// TIA Portal V16 export
// export: Created 2023-03-29T11:03:25.0566469Z, ExportSetting WithDefaults, DisplayName Totally Integrated Automation Portal, DisplayVersion V16 Update 6, DisplayName TIA Portal Version Control Interface, DisplayVersion V16 Update 2, DisplayName TIA Portal Openness, DisplayVersion V16 Update 6, DisplayName STEP 7 Professional, DisplayVersion V16 Update 6, DisplayName STEP 7 Safety, DisplayVersion V16, DisplayName WinCC Advanced, DisplayVersion V16 Update 6
FUNCTION_BLOCK "Client_ModbusTCP_read_control"   // FB1, LAD
TITLE = Pobieranie parametrów sterowania
{ S7_Optimized_Access := 'TRUE' }
AUTHOR : rtecmer
VERSION : 0.1
// funkcja pobiera z servera dane przekazywanie z PLC 1 do kontroli systemu
// stored: AutoNumber true, IsIECCheckEnabled false, IsRetainMemResEnabled false, MemoryReserve 250, SetENOAutomatically false, UDAEnableTagReadback false
   VAR_IN_OUT
      modbustcp_przetwarzanie_In : Bool;
      modbustcp_przetwarzanie_out : Bool;
   END_VAR
   VAR_TEMP   // added for the SCL form of the ladder/FBD networks
      _w1 : Bool;
      _w2 : Bool;
   END_VAR
BEGIN

REGION Network 1: Inicjacja modbus po błędzie i restarcie
END_REGION

REGION Network 2
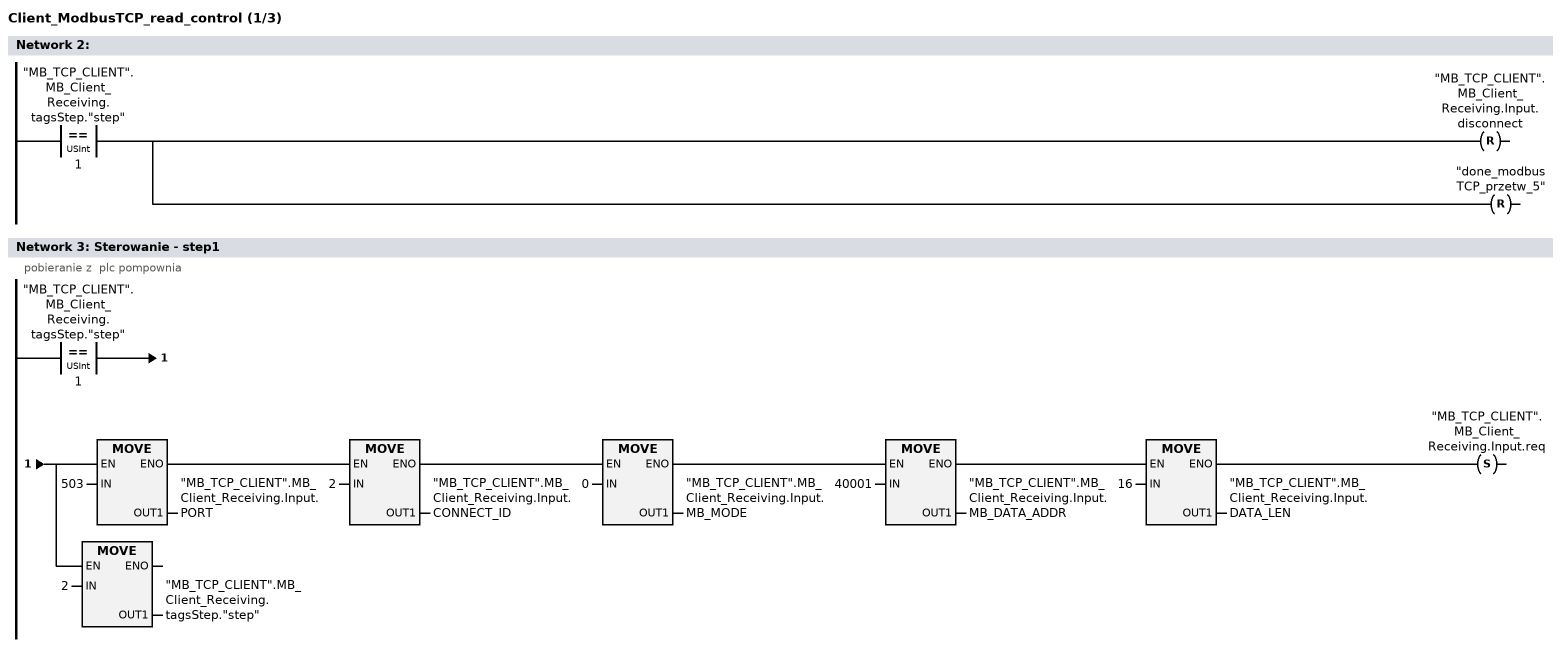
   RUNG wire#powerrail
      { S7_Templates := "SrcType := USInt" } EQ_Contact(in1 := "MB_TCP_CLIENT".MB_Client_Receiving.tagsStep."step", in2 := 1)
      wire#w1
      R_Coil( "MB_TCP_CLIENT".MB_Client_Receiving.Input.disconnect )
   END_RUNG
   RUNG wire#w1
      R_Coil( "done_modbusTCP_przetw_5" )
   END_RUNG
   // the same network as SCL:
   IF "MB_TCP_CLIENT".MB_Client_Receiving.tagsStep."step" = 1 THEN
       "MB_TCP_CLIENT".MB_Client_Receiving.Input.disconnect := FALSE;
       "done_modbusTCP_przetw_5" := FALSE;
   END_IF;
END_REGION

REGION Network 3: Sterowanie - step1
   // pobieranie z  plc pompownia
   RUNG wire#powerrail
      { S7_Templates := "SrcType := USInt" } EQ_Contact(in1 := "MB_TCP_CLIENT".MB_Client_Receiving.tagsStep."step", in2 := 1)
      wire#w1
      { S7_GenerateENO := "TRUE" } Move(in := 503, out1 => "MB_TCP_CLIENT".MB_Client_Receiving.Input.PORT)
      { S7_GenerateENO := "TRUE" } Move(in := 2, out1 => "MB_TCP_CLIENT".MB_Client_Receiving.Input.CONNECT_ID)
      { S7_GenerateENO := "TRUE" } Move(in := 0, out1 => "MB_TCP_CLIENT".MB_Client_Receiving.Input.MB_MODE)
      { S7_GenerateENO := "TRUE" } Move(in := 40001, out1 => "MB_TCP_CLIENT".MB_Client_Receiving.Input.MB_DATA_ADDR)
      { S7_GenerateENO := "TRUE" } Move(in := 16, out1 => "MB_TCP_CLIENT".MB_Client_Receiving.Input.DATA_LEN)
      S_Coil( "MB_TCP_CLIENT".MB_Client_Receiving.Input.req )
   END_RUNG
   RUNG wire#w1
      { S7_GenerateENO := "TRUE" } Move(in := 2, out1 => "MB_TCP_CLIENT".MB_Client_Receiving.tagsStep."step")
   END_RUNG
   // the same network as SCL:
   // ENO of a box is taken as its EN; it also drops when the box reports an error
   IF "MB_TCP_CLIENT".MB_Client_Receiving.tagsStep."step" = 1 THEN
       "MB_TCP_CLIENT".MB_Client_Receiving.Input.PORT := 503;
       "MB_TCP_CLIENT".MB_Client_Receiving.Input.CONNECT_ID := 2;
       "MB_TCP_CLIENT".MB_Client_Receiving.Input.MB_MODE := 0;
       "MB_TCP_CLIENT".MB_Client_Receiving.Input.MB_DATA_ADDR := 40001;
       "MB_TCP_CLIENT".MB_Client_Receiving.Input.DATA_LEN := 16;
       "MB_TCP_CLIENT".MB_Client_Receiving.Input.req := TRUE;
       "MB_TCP_CLIENT".MB_Client_Receiving.tagsStep."step" := 2;
   END_IF;
END_REGION

REGION Network 4: step 2
   // zmienne sterowania
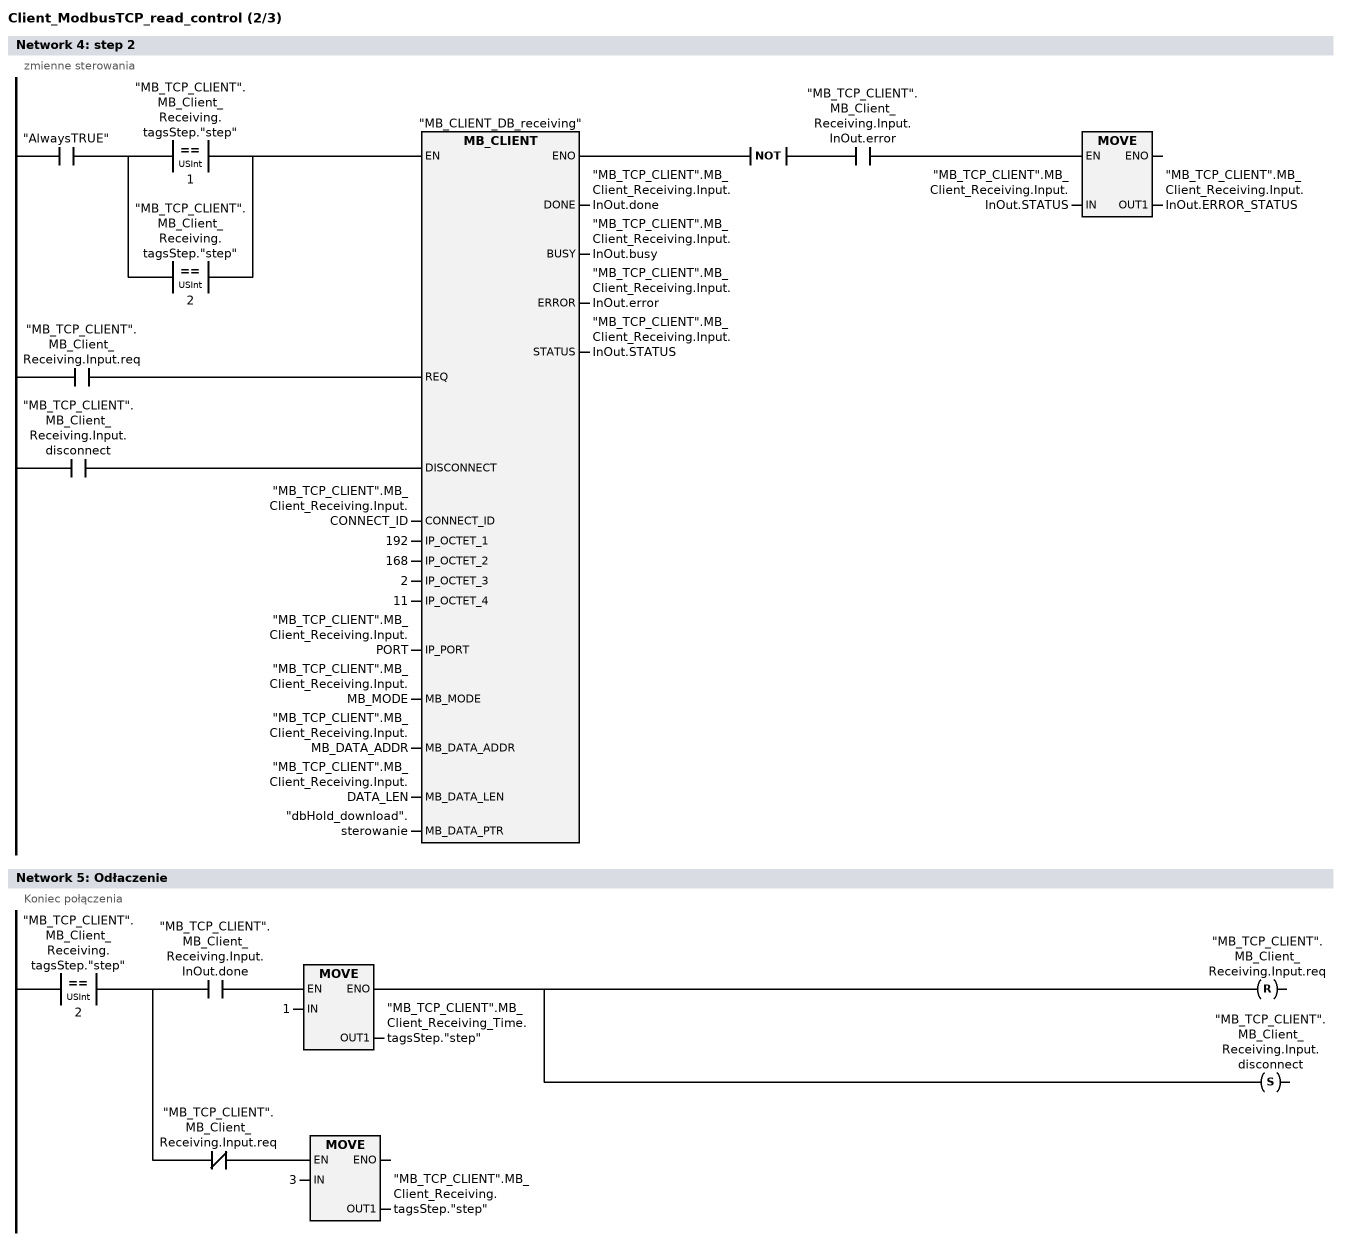
   RUNG wire#powerrail
      Contact( "AlwaysTRUE" )
      wire#w1
      { S7_Templates := "SrcType := USInt" } EQ_Contact(in1 := "MB_TCP_CLIENT".MB_Client_Receiving.tagsStep."step", in2 := 1)
      wire#w2
      { S7_Templates := "[card1200 := 1, card1500 := 0]" } "MB_CLIENT_DB_receiving".MB_CLIENT(REQ := wire#w3, DISCONNECT := wire#w4, CONNECT_ID := "MB_TCP_CLIENT".MB_Client_Receiving.Input.CONNECT_ID, IP_OCTET_1 := 192, IP_OCTET_2 := 168, IP_OCTET_3 := 2, IP_OCTET_4 := 11, IP_PORT := "MB_TCP_CLIENT".MB_Client_Receiving.Input.PORT, MB_MODE := "MB_TCP_CLIENT".MB_Client_Receiving.Input.MB_MODE, MB_DATA_ADDR := "MB_TCP_CLIENT".MB_Client_Receiving.Input.MB_DATA_ADDR, MB_DATA_LEN := "MB_TCP_CLIENT".MB_Client_Receiving.Input.DATA_LEN, MB_DATA_PTR := "dbHold_download".sterowanie, DONE => "MB_TCP_CLIENT".MB_Client_Receiving.Input.InOut.done, BUSY => "MB_TCP_CLIENT".MB_Client_Receiving.Input.InOut.busy, ERROR => "MB_TCP_CLIENT".MB_Client_Receiving.Input.InOut.error, STATUS => "MB_TCP_CLIENT".MB_Client_Receiving.Input.InOut.STATUS)
      Not()
      Contact( "MB_TCP_CLIENT".MB_Client_Receiving.Input.InOut.error )
      Move(in := "MB_TCP_CLIENT".MB_Client_Receiving.Input.InOut.STATUS, out1 => "MB_TCP_CLIENT".MB_Client_Receiving.Input.InOut.ERROR_STATUS)
   END_RUNG
   RUNG wire#w1
      { S7_Templates := "SrcType := USInt" } EQ_Contact(in1 := "MB_TCP_CLIENT".MB_Client_Receiving.tagsStep."step", in2 := 2)
   END_RUNG wire#w2
   RUNG wire#powerrail
      Contact( "MB_TCP_CLIENT".MB_Client_Receiving.Input.req )
   END_RUNG wire#w3
   RUNG wire#powerrail
      Contact( "MB_TCP_CLIENT".MB_Client_Receiving.Input.disconnect )
   END_RUNG wire#w4
   // the same network as SCL:
   #_w1 := "AlwaysTRUE" AND (("MB_TCP_CLIENT".MB_Client_Receiving.tagsStep."step" = 1) OR ("MB_TCP_CLIENT".MB_Client_Receiving.tagsStep."step" = 2));
   "MB_CLIENT_DB_receiving"(EN := #_w1,   // MB_CLIENT
                           REQ := "MB_TCP_CLIENT".MB_Client_Receiving.Input.req,
                           DISCONNECT := "MB_TCP_CLIENT".MB_Client_Receiving.Input.disconnect,
                           CONNECT_ID := "MB_TCP_CLIENT".MB_Client_Receiving.Input.CONNECT_ID,
                           IP_OCTET_1 := 192,
                           IP_OCTET_2 := 168,
                           IP_OCTET_3 := 2,
                           IP_OCTET_4 := 11,
                           IP_PORT := "MB_TCP_CLIENT".MB_Client_Receiving.Input.PORT,
                           MB_MODE := "MB_TCP_CLIENT".MB_Client_Receiving.Input.MB_MODE,
                           MB_DATA_ADDR := "MB_TCP_CLIENT".MB_Client_Receiving.Input.MB_DATA_ADDR,
                           MB_DATA_LEN := "MB_TCP_CLIENT".MB_Client_Receiving.Input.DATA_LEN,
                           MB_DATA_PTR := "dbHold_download".sterowanie,
                           DONE => "MB_TCP_CLIENT".MB_Client_Receiving.Input.InOut.done,
                           BUSY => "MB_TCP_CLIENT".MB_Client_Receiving.Input.InOut.busy,
                           ERROR => "MB_TCP_CLIENT".MB_Client_Receiving.Input.InOut.error,
                           STATUS => "MB_TCP_CLIENT".MB_Client_Receiving.Input.InOut.STATUS,
                           ENO => #_w2);
   IF NOT #_w2 AND "MB_TCP_CLIENT".MB_Client_Receiving.Input.InOut.error THEN
       "MB_TCP_CLIENT".MB_Client_Receiving.Input.InOut.ERROR_STATUS := "MB_TCP_CLIENT".MB_Client_Receiving.Input.InOut.STATUS;
   END_IF;
END_REGION

REGION Network 5: Odłaczenie
   // Koniec połączenia
   RUNG wire#powerrail
      { S7_Templates := "SrcType := USInt" } EQ_Contact(in1 := "MB_TCP_CLIENT".MB_Client_Receiving.tagsStep."step", in2 := 2)
      wire#w1
      Contact( "MB_TCP_CLIENT".MB_Client_Receiving.Input.InOut.done )
      Move(in := 1, out1 => "MB_TCP_CLIENT".MB_Client_Receiving_Time.tagsStep."step")
      wire#w2
      R_Coil( "MB_TCP_CLIENT".MB_Client_Receiving.Input.req )
   END_RUNG
   RUNG wire#w2
      S_Coil( "MB_TCP_CLIENT".MB_Client_Receiving.Input.disconnect )
   END_RUNG
   RUNG wire#w1
      I_Contact( "MB_TCP_CLIENT".MB_Client_Receiving.Input.req )
      Move(in := 3, out1 => "MB_TCP_CLIENT".MB_Client_Receiving.tagsStep."step")
   END_RUNG
   // the same network as SCL:
   #_w1 := "MB_TCP_CLIENT".MB_Client_Receiving.tagsStep."step" = 2;
   IF #_w1 AND "MB_TCP_CLIENT".MB_Client_Receiving.Input.InOut.done THEN
       "MB_TCP_CLIENT".MB_Client_Receiving_Time.tagsStep."step" := 1;
       "MB_TCP_CLIENT".MB_Client_Receiving.Input.req := FALSE;
       "MB_TCP_CLIENT".MB_Client_Receiving.Input.disconnect := TRUE;
   END_IF;
   IF #_w1 AND NOT "MB_TCP_CLIENT".MB_Client_Receiving.Input.req THEN
       "MB_TCP_CLIENT".MB_Client_Receiving.tagsStep."step" := 3;
   END_IF;
END_REGION

REGION Network 6
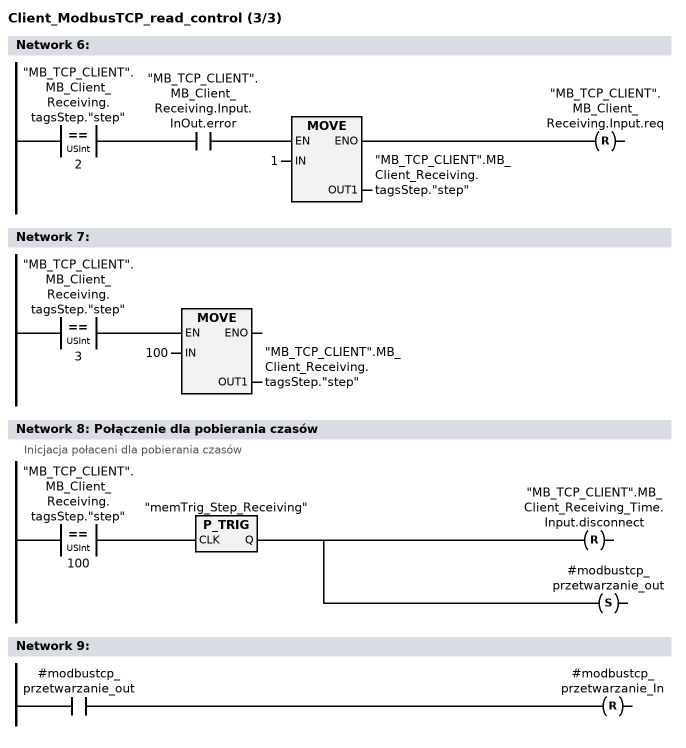
   RUNG wire#powerrail
      { S7_Templates := "SrcType := USInt" } EQ_Contact(in1 := "MB_TCP_CLIENT".MB_Client_Receiving.tagsStep."step", in2 := 2)
      Contact( "MB_TCP_CLIENT".MB_Client_Receiving.Input.InOut.error )
      Move(in := 1, out1 => "MB_TCP_CLIENT".MB_Client_Receiving.tagsStep."step")
      R_Coil( "MB_TCP_CLIENT".MB_Client_Receiving.Input.req )
   END_RUNG
   // the same network as SCL:
   #_w1 := ("MB_TCP_CLIENT".MB_Client_Receiving.tagsStep."step" = 2) AND "MB_TCP_CLIENT".MB_Client_Receiving.Input.InOut.error;
   IF #_w1 THEN
       "MB_TCP_CLIENT".MB_Client_Receiving.tagsStep."step" := 1;
       "MB_TCP_CLIENT".MB_Client_Receiving.Input.req := FALSE;
   END_IF;
END_REGION

REGION Network 7
   RUNG wire#powerrail
      { S7_Templates := "SrcType := USInt" } EQ_Contact(in1 := "MB_TCP_CLIENT".MB_Client_Receiving.tagsStep."step", in2 := 3)
      Move(in := 100, out1 => "MB_TCP_CLIENT".MB_Client_Receiving.tagsStep."step")
   END_RUNG
   // the same network as SCL:
   IF "MB_TCP_CLIENT".MB_Client_Receiving.tagsStep."step" = 3 THEN
       "MB_TCP_CLIENT".MB_Client_Receiving.tagsStep."step" := 100;
   END_IF;
END_REGION

REGION Network 8: Połączenie dla pobierania czasów
   // Inicjacja połaceni dla pobierania czasów
   RUNG wire#powerrail
      { S7_Templates := "SrcType := USInt" } EQ_Contact(in1 := "MB_TCP_CLIENT".MB_Client_Receiving.tagsStep."step", in2 := 100)
      P_Trig( "memTrig_Step_Receiving" )
      wire#w1
      R_Coil( "MB_TCP_CLIENT".MB_Client_Receiving_Time.Input.disconnect )
   END_RUNG
   RUNG wire#w1
      S_Coil( #modbustcp_przetwarzanie_out )
   END_RUNG
   // the same network as SCL:
   #_w1 := "MB_TCP_CLIENT".MB_Client_Receiving.tagsStep."step" = 100;
   #_w2 := #_w1 AND NOT "memTrig_Step_Receiving";   // rising edge
   "memTrig_Step_Receiving" := #_w1;
   IF #_w2 THEN
       "MB_TCP_CLIENT".MB_Client_Receiving_Time.Input.disconnect := FALSE;
       #modbustcp_przetwarzanie_out := TRUE;
   END_IF;
END_REGION

REGION Network 9
   RUNG wire#powerrail
      Contact( #modbustcp_przetwarzanie_out )
      R_Coil( #modbustcp_przetwarzanie_In )
   END_RUNG
   // the same network as SCL:
   IF #modbustcp_przetwarzanie_out THEN #modbustcp_przetwarzanie_In := FALSE; END_IF;
END_REGION
END_FUNCTION_BLOCK
